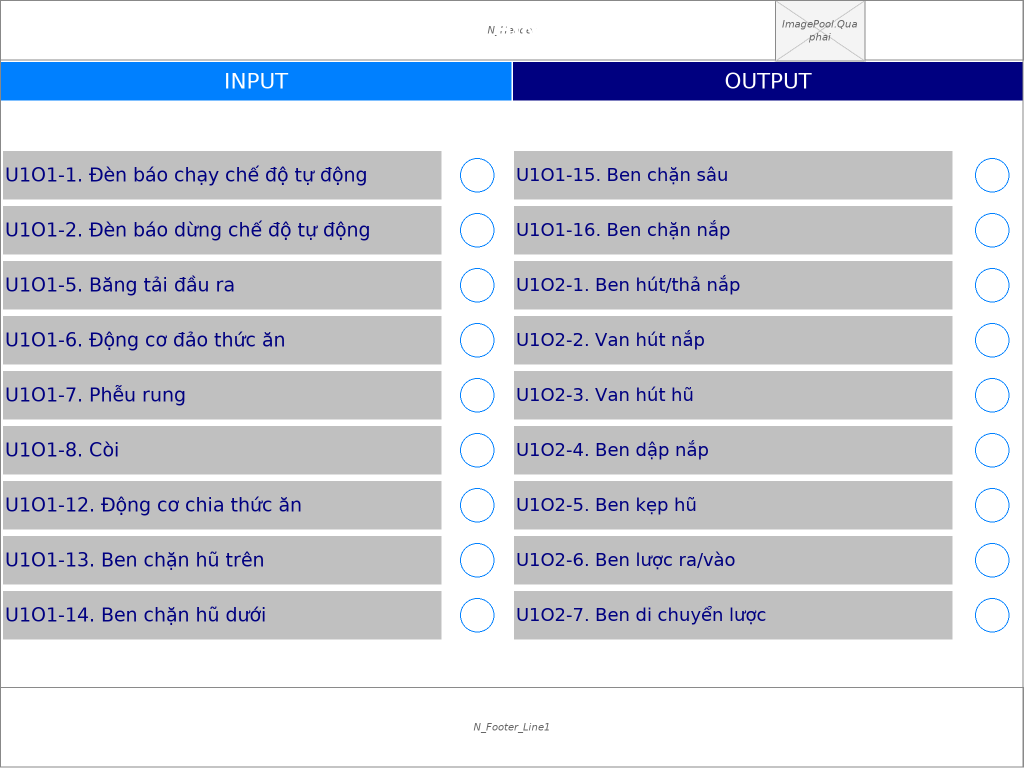
VISUALIZATION N_PLC_O1  // 1024x768
    Frame (0,687 1024x80)
        shows N_Footer_Line1()
    Frame (0,0 1024x60)
        shows N_Header()
    Textfield (353,5 400x50), "MÀN HÌNH IO LINE 1"
    Rectangle (0,61 512x40), "INPUT"
        OnMouseClick: change screen: N_PLC_I1
    Rectangle (512,61 512x40), "OUTPUT"
        OnMouseClick: change screen: N_PLC_O1
    Image (775,0 90x61), image: ImagePool.Qua phai
        OnMouseClick: change screen: N_PLC_O2
    Rectangle (2,150 440x50), "U1O1-1. Đèn báo chạy chế độ tự động"
    Rectangle (2,205 440x50), "U1O1-2. Đèn báo dừng chế độ tự động"
    Rectangle (2,260 440x50), "U1O1-5. Băng tải đầu ra"
    Ellipse (460,158 34x34), colour toggle: GVL_IO.bLight_Running, input disabled if: true
    Ellipse (460,213 34x34), colour toggle: GVL_IO.bLight_Stop, input disabled if: true
    Rectangle (2,315 440x50), "U1O1-6. Động cơ đảo thức ăn"
    Rectangle (2,370 440x50), "U1O1-7. Phễu rung"
    Rectangle (2,425 440x50), "U1O1-8. Còi"
    Rectangle (2,480 440x50), "U1O1-12. Động cơ chia thức ăn"
    Rectangle (2,535 440x50), "U1O1-13. Ben chặn hũ trên"
    Rectangle (2,590 440x50), "U1O1-14. Ben chặn hũ dưới"
    Rectangle (513,150 440x50), "U1O1-15. Ben chặn sâu"
    Rectangle (513,205 440x50), "U1O1-16. Ben chặn nắp"
    Ellipse (460,268 34x34), colour toggle: PR_Conveyor_Out.fb_Conveyor.fbInverter.bVFD, input disabled if: true
    Ellipse (460,323 34x34), colour toggle: PR_Line01.fb_FoodMixer.fbInverter.bVFD, input disabled if: true
    Ellipse (460,378 34x34), colour toggle: PR_Line01.fb_WormWeight.fbInverter.bVFD, input disabled if: true
    Ellipse (460,433 34x34), colour toggle: GVL_IO.bSirens, input disabled if: true
    Ellipse (460,488 34x34), colour toggle: PR_Line01.fb_FoodWeight.fbDriver.bVFD, input disabled if: true
    Ellipse (460,543 34x34), colour toggle: PR_Line01.fb_CupSupply.fbCylinder_Up.bMoveExtend, input disabled if: true
    Ellipse (460,598 34x34), colour toggle: PR_Line01.fb_CupSupply.fbCylinder_Dw.bMoveRetract, input disabled if: true
    Ellipse (975,158 34x34), colour toggle: PR_Line02.fb_WormWeight.fbCylinder.bMoveRetract, input disabled if: true
    Ellipse (975,213 34x34), colour toggle: PR_Line01.fb_LidSupply.fbCylinder_LidStopper.bMoveRetract, input disabled if: true
    Rectangle (513,260 440x50), "U1O2-1. Ben hút/thả nắp"
    Ellipse (975,268 34x34), colour toggle: PR_Line02.fb_LidSupply.fbCylinder_Suction.bMoveExtend, input disabled if: true
    Rectangle (513,315 440x50), "U1O2-2. Van hút nắp"
    Rectangle (513,370 440x50), "U1O2-3. Van hút hũ"
    Rectangle (513,425 440x50), "U1O2-4. Ben dập nắp"
    Rectangle (513,480 440x50), "U1O2-5. Ben kẹp hũ"
    Rectangle (513,535 440x50), "U1O2-6. Ben lược ra/vào"
    Rectangle (513,590 440x50), "U1O2-7. Ben di chuyển lược"
    Ellipse (975,323 34x34), colour toggle: PR_Line02.fb_LidSupply.fbLidSuctionValve.bSuck, input disabled if: true
    Ellipse (975,378 34x34), colour toggle: PR_Line02.fb_LidSupply.fbCupSuctionValve.bSuck, input disabled if: true
    Ellipse (975,433 34x34), colour toggle: PR_Line02.fb_LidClose.fbCylinder_LidClose.bMoveExtend, input disabled if: true
    Ellipse (975,488 34x34), colour toggle: PR_Line01.fb_Transfer.fbCylinder_Clip.bMoveRetract, input disabled if: true
    Ellipse (975,543 34x34), colour toggle: PR_Line01.fb_Transfer.fbCylinder_Comb.bMoveExtend, input disabled if: true
    Ellipse (975,598 34x34), colour toggle: PR_Line01.fb_Transfer.fbCylinder_Move_Comb.bMoveExtend, input disabled if: true
END_VISUALIZATION

(* stored: Version 1.1.0.1, ProductVersion 3.1.4024.12
   Visu N_PLC_O1: Id {88840a11-3df8-4a4c-b04e-c3f9c1a2ef70} *)
